// TIA Portal project "babu_motorFwdReverseHMI" (V15)

(* hardware
DEVICE "S7-1200 station_1"  S7-1200 Station
   slot 0: "Rack_0"  S7-1200 Rack  Rack  V1.0
   slot 1: "PLC_1"  CPU 1214C DC/DC/DC  6ES7 214-1AG40-0XB0  V4.2
DEVICE "HMI_1"  KTP400 Basic color PN
   slot 0: "HMI_1"  KTP400 Basic color PN  6AV6 647-0AK11-3AX0  12.0.0.0
   slot 1: "HMI_RT_1"  KTP400 Basic color PN  6AV6 647-0AK11-3AX0  12.0.0.0
   slot 5: "HMI_1.IE_CP_1"  PROFINET Interface  12.0.0.0
      slot 1: "PROFINET Interface_1"  PROFINET Interface
         slot 1: "Port_1"  Port
*)

// ===== PLC "PLC_1"  CPU 1214C DC/DC/DC =====

VAR_GLOBAL   // PLC tag table "Default tag table"
   "START PB" AT %M0.0 : Bool;
   "MOTOR ON MEM" AT %M0.1 : Bool;
   "STOP" AT %M0.2 : Bool;
   "START PB MEM" AT %M0.3 : Bool;
   "STOP PB MEM" AT %M0.4 : Bool;
   "FWD PB" AT %M0.5 : Bool;
   "FWD PB MEM" AT %M0.6 : Bool;
   "REV PB" AT %M0.7 : Bool;
   "REV PB MEM" AT %M1.0 : Bool;
   "MOTOR FORWARD" AT %Q0.0 : Bool;
   "MOTOR REVERSE" AT %Q0.1 : Bool;
END_VAR

ORGANIZATION_BLOCK "Main"   // OB1, LAD, ProgramCycle
TITLE = "Main Program Sweep (Cycle)"
{ S7_Optimized_Access := 'TRUE' }
VERSION : 0.1
   VAR_INPUT
      Initial_Call : Bool;   // Initial call of this OB
      Remanence : Bool;   // =True, if remanent data are available
   END_VAR
   VAR_TEMP   // added for the SCL form of the ladder/FBD networks
      _w1 : Bool;
      _w2 : Bool;
      _w3 : Bool;
      _w4 : Bool;
   END_VAR
BEGIN

REGION Network 1
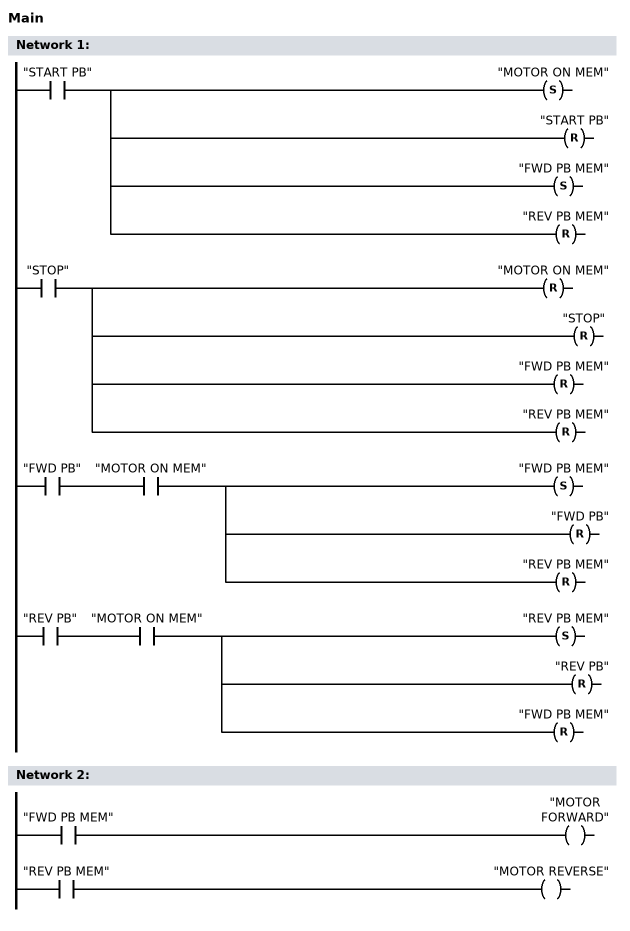
   RUNG wire#powerrail
      Contact( "START PB" )
      wire#w1
      S_Coil( "MOTOR ON MEM" )
   END_RUNG
   RUNG wire#w1
      R_Coil( "START PB" )
   END_RUNG
   RUNG wire#w1
      S_Coil( "FWD PB MEM" )
   END_RUNG
   RUNG wire#w1
      R_Coil( "REV PB MEM" )
   END_RUNG
   RUNG wire#powerrail
      Contact( "STOP" )
      wire#w2
      R_Coil( "MOTOR ON MEM" )
   END_RUNG
   RUNG wire#w2
      R_Coil( "STOP" )
   END_RUNG
   RUNG wire#w2
      R_Coil( "FWD PB MEM" )
   END_RUNG
   RUNG wire#w2
      R_Coil( "REV PB MEM" )
   END_RUNG
   RUNG wire#powerrail
      Contact( "FWD PB" )
      Contact( "MOTOR ON MEM" )
      wire#w3
      S_Coil( "FWD PB MEM" )
   END_RUNG
   RUNG wire#w3
      R_Coil( "FWD PB" )
   END_RUNG
   RUNG wire#w3
      R_Coil( "REV PB MEM" )
   END_RUNG
   RUNG wire#powerrail
      Contact( "REV PB" )
      Contact( "MOTOR ON MEM" )
      wire#w4
      S_Coil( "REV PB MEM" )
   END_RUNG
   RUNG wire#w4
      R_Coil( "REV PB" )
   END_RUNG
   RUNG wire#w4
      R_Coil( "FWD PB MEM" )
   END_RUNG
   // the same network as SCL:
   IF "START PB" THEN "MOTOR ON MEM" := TRUE; END_IF;
   #_w1 := "START PB";
   IF #_w1 THEN
       "START PB" := FALSE;
       "FWD PB MEM" := TRUE;
       "REV PB MEM" := FALSE;
   END_IF;
   IF "STOP" THEN "MOTOR ON MEM" := FALSE; END_IF;
   #_w2 := "STOP";
   IF #_w2 THEN
       "STOP" := FALSE;
       "FWD PB MEM" := FALSE;
       "REV PB MEM" := FALSE;
   END_IF;
   IF "FWD PB" AND "MOTOR ON MEM" THEN "FWD PB MEM" := TRUE; END_IF;
   #_w3 := "FWD PB" AND "MOTOR ON MEM";
   IF #_w3 THEN
       "FWD PB" := FALSE;
       "REV PB MEM" := FALSE;
   END_IF;
   IF "REV PB" AND "MOTOR ON MEM" THEN "REV PB MEM" := TRUE; END_IF;
   #_w4 := "REV PB" AND "MOTOR ON MEM";
   IF #_w4 THEN
       "REV PB" := FALSE;
       "FWD PB MEM" := FALSE;
   END_IF;
END_REGION

REGION Network 2
   RUNG wire#powerrail
      Contact( "FWD PB MEM" )
      Coil( "MOTOR FORWARD" )
   END_RUNG
   RUNG wire#powerrail
      Contact( "REV PB MEM" )
      Coil( "MOTOR REVERSE" )
   END_RUNG
   // the same network as SCL:
   "MOTOR FORWARD" := "FWD PB MEM";
   "MOTOR REVERSE" := "REV PB MEM";
END_REGION
END_ORGANIZATION_BLOCK

(* ===== HMI "HMI_RT_1" =====
system functions are stored by id; their names below are inferred from use
connection "HMI_Connection_1": ETHERNET, SMART_S7_1200_OMS
connection "HMI_Connection_2": ETHERNET, SMART_S7_1200_OMS

HMI tags "Default tag table"
   "START PB" : Bool = PLC "START PB" AT %M0.0, 1 s
   "STOP" : Bool = PLC STOP AT %M0.2, 1 s
   "MOTOR FORWARD" : Bool = PLC "MOTOR FORWARD" AT %Q0.0, 1 s
   "FWD PB MEM" : Bool = PLC "FWD PB MEM" AT %M0.6, 1 s
   "REV PB MEM" : Bool = PLC "REV PB MEM" AT %M1.0, 1 s
   "MOTOR ON MEM" : Bool = PLC "MOTOR ON MEM" AT %M0.1, 1 s
   "FWD PB" : Bool = PLC "FWD PB" AT %M0.5, 1 s
   "REV PB" : Bool = PLC "REV PB" AT %M0.7, 1 s

screen "Screen_1" 480x272
   Circle "Circle_3" at 186,141 size 99x99
      Visibility <- "MOTOR ON MEM"
   Button "Button_1" at 106,15 size 96x32; TextOff 'START'; TextOn 'STARTED'
      on Press: SetBit("START PB")
      on Release: ResetBit("START PB")
      Appearance <- "START PB"
   Button "Button_2" at 106,73 size 96x32; TextOff 'STOP'
      on Press: SetBit("STOP")
      on Release: ResetBit("STOP")
      Appearance <- "STOP"
   Button "Button_3" at 270,15 size 96x32; TextOff 'FWD...'
      on Press: SetBit("FWD PB")
      on Release: ResetBit("FWD PB")
      Appearance <- "FWD PB MEM"
   Button "Button_4" at 270,73 size 96x32; TextOff 'REV...'
      on Press: SetBit("REV PB")
      on Release: ResetBit("REV PB")
      Appearance <- "REV PB MEM"
   Circle "Circle_1" at 186,141 size 99x99
      Appearance <- "MOTOR FORWARD"
      Visibility <- "FWD PB MEM"
   TextField "Text field_2" at 306,150 size 142x20; Text '1. RED MOTOR FWD'
   TextField "Text field_3" at 306,168 size 154x20; Text '2. GREEN MOTOR REV'
   Circle "Circle_2" at 186,141 size 99x99
      Visibility <- "REV PB MEM"
   TextField "Text field_4" at 307,187 size 163x20; Text '3. YELLO MOTOR STOP'
   TextField "Text field_1" at 209,177 size 55x20; Text 'MOTOR'
*)